// TIA Portal V20 export
TYPE "type_emRelations_em4_cmStatus"
// stored: Access Published, Namespace Unit1
   STRUCT
      SideTapeSafetyPin : "LBC_typeDigitalSignalControlNode";
      SideTapeJRDetect : "LBC_typeDigitalSignalControlNode";
      SideTapeDiameter : "LBC_typeDigitalSignalControlNode";
      SideTapeFixStageAxisX : "LBC_typeAxis64PosControlNode";
      SideTapeFixStageAxisC : "LBC_typeAxis64PosControlNode";
      SideTapeAttachmentAxisX : "LBC_typeAxis64PosControlNode";
      SideTapeAttachmentAxisY : "LBC_typeAxis64PosControlNode";
      SideTapeLoadingDownUp : "LBC_typeTwoWayActuatorControlNode";
      SideTapeLoadingClampOpenClose : "LBC_typeTwoWayActuatorControlNode";
      SideTapeCutterBwdFwd : "LBC_typeTwoWayActuatorControlNode";
      SideTapeCutterClampBwdFwd : "LBC_typeTwoWayActuatorControlNode";
      SideTapeTensionBwdFwd : "LBC_typeTwoWayActuatorControlNode";
      SideTapeAttachmentLeftBwdFwd : "LBC_typeTwoWayActuatorControlNode";
      SideTapeAttachmentRightBwdFwd : "LBC_typeTwoWayActuatorControlNode";
      SideTapeAttachmentBtmBwdFwd : "LBC_typeTwoWayActuatorControlNode";
      SideTapeFixStageClampOpenClose : "LBC_typeTwoWayActuatorControlNode";
      SideTapeAttachment1TopVaccumOffOn : "LBC_typeTwoWayActuatorControlNode";
      SideTapeAttachment1BtmVaccumOffOn : "LBC_typeTwoWayActuatorControlNode";
      SideTapeAttachment2TopVaccumOffOn : "LBC_typeTwoWayActuatorControlNode";
      SideTapeAttachment2BtmVaccumOffOn : "LBC_typeTwoWayActuatorControlNode";
      QrHandyReader : "LER_typeDM8700ControlNode";
   END_STRUCT;
END_TYPE
